// SIMATIC S7-200 project (STEP 7-Micro/WIN), CPU 221 REL 01.10

SYMBOL_TABLE IO
急停按钮             I0.0
自动/手动            I0.1
启动按钮             I0.2
复位按钮             I0.4
标准气缸后退检测-L       I0.5
流水线顶升气缸下降检测      I0.7
流水线顶升气缸上升检测      I1.0
上工位检测            I1.1
导杆气缸后退检测         I1.2
标准气缸前进检测-R       I1.3
标准气缸后退检测-R       I1.5
电动缸SRDY          I2.0
电动缸STOP          I2.1
电动缸ALRM          I2.2
输入轴SRDY          I2.3
输入轴STOP          I2.4
输入轴ALRM          I2.5
导杆气缸前进检测         I2.6
标准气缸前进检测-L       I2.7
本工位检测            I3.6
下工位检测            I3.7
电动缸上电            Q0.0
输入轴上电            Q0.1
电动缸急停            Q0.2
输入轴急停            Q0.3
红灯               Q0.4
黄灯               Q0.5
绿灯               Q0.6
蜂鸣器              Q0.7
顶升气缸上位顶升         Q1.0
顶升气缸上位下降         Q1.1
本工位放行            Q2.0
上工位放行            Q2.1
标准气缸后退-R         Q2.2
标准气缸前进-L         Q2.3
导杆气缸前进           Q2.4
标准气缸前进-R         Q2.5
导杆气缸后退           Q3.0
标准气缸后退-L         Q3.1
END_SYMBOL_TABLE

SYMBOL_TABLE M3000
流水线工步号           MW3000
产品类型             MW3002
RFID工步号          MW3004
芯片编号             MW3006
一键初始化工步号         MW3008
通讯状态             M3010.0
本工位合格            M3010.1
本工位完成            M3010.2
不合格报警            M3010.3
RFID读取触发         M3010.4
RFID读取完成         M3010.5
RFID运行中          M3010.6
M一键初始化按钮         M3011.0
M一键初始化完成         M3011.1
M上工位放行           M3020.0
M本工位放行           M3020.1
M流水线顶升顶升         M3020.2
M流水线顶升下降         M3020.3
M导杆气缸前进          M3021.0
M导杆气缸后退          M3021.1
M标准气缸后退-L        M3021.2
M标准气缸前进-L        M3021.3
M标准气缸后退-R        M3021.4
M标准气缸前进-R        M3021.5
上工位合格            M3030.0
上工位完成            M3030.1
联线状态             M3040.0
报警工步号            MW3050
员工权限             M3060.0
电动缸工步号           MW3100
M流水线准备好信号(交互)    M3110.0
M电动缸自动完成信号(交     M3110.1
END_SYMBOL_TABLE
